FUNCTION "Main sensori" : Void
{ S7_Optimized_Access := 'TRUE' }
VERSION : 0.1
   VAR_INPUT
      K_Sensore : Int;
      K_Zona : Int;
   END_VAR

   VAR_TEMP
      K_SensoreInt : Int;
      K_ZonaInt : Int;
   END_VAR


BEGIN
END_FUNCTION

